Fanuc KAREL source: kt00295.KL

-- PROVISIONAL review KL for V940-1; original PC SHA256 0318c5416d591ae9d3ce69395c04d604bd09ff1a9829935c8fd7493f21e73766
-- Incomplete behavior may be omitted. Consult companion uncertainty JSON. Do not deploy.
PROGRAM KT00295
%NOLOCKGROUP
VAR
  I1 : INTEGER
  OUT : BOOLEAN
-- UNRESOLVED_DECL Y2 type=002018
BEGIN
  -- V9_ZERO_TABLE_METADATA_HINT layout=0001; no indexed target words; source/name/runtime held
  -- UNRESOLVED_PC offsets 5-16; opcodes 2E,23
  -- UNRESOLVED_PC offsets 21-35; opcodes 2E,22,9D,33,B2
  -- UNRESOLVED_PC offsets 40-62; opcodes 21,22,9D,33,B1,58,23
  -- UNRESOLVED_PC offsets 67-71; opcodes 7F
END KT00295
